FUNCTION_BLOCK PUBLIC RoutePlanner
VAR_INPUT
END_VAR
VAR_OUTPUT
END_VAR
VAR
	RejecLoadPosChoice			:       UINT :=5;
	RejectNextStationLocation	:		REAL;
	RejectNextStationIndex		:		BYTE;
	
	GoodULPosChoice				:       UINT :=5;
	GoodULNextStationLocation	:		REAL;
	GoodULNextStationIndex		:		BYTE;
	GoodFullCount : UINT := 0;
	PremiumFullCount : UINT := 0;
	GoodUL_1_NextStationFlag : BYTE := 5; // Next Station is defaulted to 5 ( reject)
	GoodUL_2_NextStationFlag : BYTE := 5; // Next Station is defaulted to 5 ( reject)
	GoodUL_3_NextStationFlag : BYTE := 5; // Next Station is defaulted to 5 ( reject)
	GoodUL_4_NextStationFlag : BYTE := 5; // Next Station is defaulted to 5 ( reject)
END_VAR

;

METHOD PUBLIC M_ExitCapInsertSta : BOOL
VAR_INPUT
	VehicleID		:	BYTE;
END_VAR
IF (PartsData.Status[VehicleID].OverallStatus <> ePartStatus.eReject AND 
    PartsData.Status[VehicleID].OverallStatus <> ePartStatus.eEmpty ) THEN  // we have a good part
   IF (LotsData.Lot.GoodUnloadEnabled) THEN // Good Unload is Enabled
		MoveToGoodUnload(VehicleID);
	ELSE // just go to reject
		MoveToReject(VehicleID);		
	END_IF		
ELSE  // we have a reject	
	MoveToReject(VehicleID);			
END_IF



(*

IF (PartsData.Status[VehicleID].OverallStatus = ePartStatus.eCapInserted) THEN
	Stations.fbVehicleManager[VehicleID].M_SetNextMoveParams(Pos:= MM_CONST.GOOD_UNLOAD_POS, Vel := 2.0, Acc := 2.0, StationIndex := MM_CONST.GOOD_UNLOAD_STA );
	Stations.fbVehicleManager[VehicleID].TriggerVehMov := TRUE;
ELSE 
	Stations.fbVehicleManager[VehicleID].M_SetNextMoveParams(Pos:= MM_CONST.REJECT_ULOAD_POS, Vel := 2.0, Acc := 2.0, StationIndex := MM_CONST.REJECT_ULOAD_STA );
 	Stations.fbVehicleManager[VehicleID].TriggerVehMov := TRUE;		
END_IF
*)

(*
Stations.fbVehicleManager[VehicleID].M_SetNextMoveParams(Pos:= MM_CONST.REJECT_ULOAD_POS, Vel := 2.0, Acc := 2.0, StationIndex := MM_CONST.REJECT_ULOAD_STA );
Stations.fbVehicleManager[VehicleID].TriggerVehMov := TRUE;
*)
END_METHOD

METHOD PUBLIC M_ExitGoodUnload : BOOL
VAR_INPUT
	VehicleID		:	BYTE;
END_VAR
MoveToReject(VehicleID);
END_METHOD

METHOD PUBLIC M_ExitGoodUnload_1 : BOOL
VAR_INPUT
	VehicleID		:	BYTE;
END_VAR
CASE GoodUL_1_NextStationFlag OF
	
    2:	
		MoveToGoodUnload_2(VehicleID);	
	
    3:
		MoveToGoodUnload_3(VehicleID);	
	
    4:
		MoveToGoodUnload_4(VehicleID);	
 
ELSE
		 MoveToReject(VehicleID);
	
END_CASE;
END_METHOD

METHOD PUBLIC M_ExitGoodUnload_2 : BOOL
VAR_INPUT
	VehicleID		:	BYTE;
END_VAR
CASE GoodUL_2_NextStationFlag OF
	
	
    3:
		MoveToGoodUnload_3(VehicleID);	
	
    4:
		MoveToGoodUnload_4(VehicleID);	
 
ELSE
		 MoveToReject(VehicleID);
	
END_CASE;
END_METHOD

METHOD PUBLIC M_ExitGoodUnload_3 : BOOL
VAR_INPUT
	VehicleID		:	BYTE;
END_VAR
CASE GoodUL_3_NextStationFlag OF
	

    4:
		MoveToGoodUnload_4(VehicleID);	
 
ELSE
		 MoveToReject(VehicleID);
	
END_CASE;
END_METHOD

METHOD PUBLIC M_ExitGoodUnload_4 : BOOL
VAR_INPUT
	VehicleID		:	BYTE;
END_VAR
MoveToReject(VehicleID);
END_METHOD

METHOD PUBLIC M_ExitIB_StopRobotClear : BOOL
VAR_INPUT
	VehicleID		:	BYTE;
END_VAR
IF (PartsData.Status[VehicleID].OverallStatus <> ePartStatus.eReject AND 
    PartsData.Status[VehicleID].OverallStatus <> ePartStatus.eEmpty ) THEN  // we have a good part
   IF (LotsData.Lot.CapInsertEnabled) THEN // Cap Is Enabled
		MoveToCap(VehicleID);
	ELSIF (LotsData.Lot.GoodUnloadEnabled) THEN // Good Unload is Enabled
		MoveToGoodUnload(VehicleID);
	ELSE // just go to reject
		MoveToReject(VehicleID);		
	END_IF		
ELSE  // we have a reject	
	MoveToReject(VehicleID);			
END_IF
END_METHOD

METHOD PUBLIC M_ExitLoad1Sta : BOOL
VAR_INPUT
	VehicleID		:	BYTE;
END_VAR
MoveToVision(VehicleID);
//MoveToStopBeforeVision(VehicleID);
END_METHOD

METHOD PUBLIC M_ExitLoad2Sta : BOOL
VAR_INPUT
	VehicleID		:	BYTE;
END_VAR
MoveToVision(VehicleID);
//MoveToStopBeforeVision(VehicleID);
END_METHOD

METHOD PUBLIC M_ExitLoad3Sta : BOOL
VAR_INPUT
	VehicleID		:	BYTE;
END_VAR
MoveToVision(VehicleID);
//MoveToStopBeforeVision(VehicleID);
END_METHOD

METHOD PUBLIC M_ExitLoad4Sta : BOOL
VAR_INPUT
	VehicleID		:	BYTE;
END_VAR
MoveToVision(VehicleID);
//MoveToStopBeforeVision(VehicleID);
END_METHOD

METHOD PUBLIC M_ExitPistonInsertSta : BOOL
VAR_INPUT
	VehicleID		:	BYTE;
END_VAR
IF (PartsData.Status[VehicleID].OverallStatus <> ePartStatus.eReject AND 
    PartsData.Status[VehicleID].OverallStatus <> ePartStatus.eEmpty ) THEN  // we have a good part
    IF (Stations.fbLoad1Sta.HoldVehicle_IBStop) THEN //Yushin wants to load 
		MoveToIBStopRobotClear(VehicleID);
	ELSIF (LotsData.Lot.CapInsertEnabled) THEN // Cap Is Enabled
		MoveToCap(VehicleID);
	ELSIF (LotsData.Lot.GoodUnloadEnabled) THEN // Good Unload is Enabled
		MoveToGoodUnload(VehicleID);
	ELSE // just go to reject
		MoveToReject(VehicleID);		
	END_IF		
ELSE  // we have a reject	
	IF (Stations.fbLoad1Sta.HoldVehicle_IBStop) THEN //Yushin wants to load 
		MoveToIBStopRobotClear(VehicleID);
	ELSE  // just go to reject
		MoveToReject(VehicleID);			
	END_IF
END_IF

(*
IF (Stations.fbLoad1Sta.HoldVehicle_IBStop) THEN //Yushin wants to load 
	Stations.fbVehicleManager[VehicleID].M_SetNextMoveParams(Pos:= MM_CONST.IB_STOP_ROBOT_CLEAR_POS, Vel := 2.0, Acc := 2.0, StationIndex := MM_CONST.IB_STOP_ROBOT_CLEAR_STA );
	Stations.fbVehicleManager[VehicleID].TriggerVehMov := TRUE;
ELSE // move straight to the cap station or reject based on part status
    IF (PartsData.Status[VehicleID].OverallStatus = ePartStatus.ePistonInserted) THEN
		 Stations.fbVehicleManager[VehicleID].M_SetNextMoveParams(Pos:= MM_CONST.CAP_POS, Vel := 2.0, Acc := 2.0, StationIndex := MM_CONST.CAP_STA );
		 Stations.fbVehicleManager[VehicleID].TriggerVehMov := TRUE;
	ELSE 
		Stations.fbVehicleManager[VehicleID].M_SetNextMoveParams(Pos:= MM_CONST.REJECT_ULOAD_POS, Vel := 2.0, Acc := 2.0, StationIndex := MM_CONST.REJECT_ULOAD_STA );
 		Stations.fbVehicleManager[VehicleID].TriggerVehMov := TRUE;
	END_IF
   
END_IF



//Stations.fbVehicleManager[VehicleID].M_SetNextMoveParams(Pos:= MM_CONST.CAP_POS, Vel := 2.0, Acc := 2.0, StationIndex := MM_CONST.CAP_STA );
//Stations.fbVehicleManager[VehicleID].TriggerVehMov := TRUE;


// Stations.fbVehicleManager[VehicleID].M_SetNextMoveParams(Pos:= MM_CONST.REJECT_ULOAD_POS, Vel := 2.0, Acc := 2.0, StationIndex := MM_CONST.REJECT_ULOAD_STA );
 // Stations.fbVehicleManager[VehicleID].TriggerVehMov := TRUE;


(*

	Stations.fbVehicleManager[VehicleID].M_SetNextMoveParams(Pos:= MM_CONST.PISTON_POS, Vel := 2.0, Acc := 2.0, StationIndex := MM_CONST.PISTON_STA );
	Stations.fbVehicleManager[VehicleID].TriggerVehMov := TRUE;
	*)

(*


IF (Stations.fbLoad1Sta.HoldVehicle_IBStop) THEN //Yushin wants to load 
	Stations.fbVehicleManager[VehicleID].M_SetNextMoveParams(Pos:= MM_CONST.IB_STOP_ROBOT_CLEAR_POS, Vel := 2.0, Acc := 2.0, StationIndex := MM_CONST.IB_STOP_ROBOT_CLEAR_STA );
	Stations.fbVehicleManager[VehicleID].TriggerVehMov := TRUE;
ELSE // move straight to the cap station
	// NEED TO REMOVE THIS AFTER DEBUG ON 3/19/2017... WE ARE BYPASSING CAP STATION FOR NOW 
    //Stations.fbVehicleManager[VehicleID].M_SetNextMoveParams(Pos:= MM_CONST.CAP_POS, Vel := 2.0, Acc := 2.0, StationIndex := MM_CONST.CAP_STA );
	//Stations.fbVehicleManager[VehicleID].TriggerVehMov := TRUE;
	
	Stations.fbVehicleManager[VehicleID].M_SetNextMoveParams(Pos:= MM_CONST.GOOD_UNLOAD_POS, Vel := 2.0, Acc := 2.0, StationIndex := MM_CONST.GOOD_UNLOAD_STA );
	Stations.fbVehicleManager[VehicleID].TriggerVehMov := TRUE;
			
END_IF

*)
*)
END_METHOD

METHOD PUBLIC M_ExitRejectUnload : BOOL
VAR_INPUT	
	VehicleID		:	BYTE;
END_VAR
RejecLoadPosChoice := RejecLoadPosChoice -1; //we initialize with this variable as 5;
IF (RejecLoadPosChoice<=0 OR RejecLoadPosChoice>=4 ) THEN 
	RejecLoadPosChoice := 4;
END_IF
CASE RejecLoadPosChoice OF
				4: 
					RejectNextStationLocation := MM_CONST.OB_STOP_ROBOT_CLEAR_POS;
					RejectNextStationIndex	:= MM_CONST.OB_STOP_ROBOT_CLEAR_STA;
				3:
					RejectNextStationLocation := MM_CONST.LOAD_3_POS;
					RejectNextStationIndex	:= MM_CONST.LOAD_3_STA;
				2:
					RejectNextStationLocation := MM_CONST.LOAD_2_POS;
					RejectNextStationIndex	:= MM_CONST.LOAD_2_STA;
				1:
					RejectNextStationLocation := MM_CONST.LOAD_1_POS;
					RejectNextStationIndex	:= MM_CONST.LOAD_1_STA;						
END_CASE				
	
Stations.fbVehicleManager[VehicleID].M_SetNextMoveParams(Pos:= RejectNextStationLocation, Vel := 2.0, Acc := 2.0, StationIndex := RejectNextStationIndex );
Stations.fbVehicleManager[VehicleID].TriggerVehMov := TRUE;
END_METHOD

METHOD PUBLIC M_ExitVisionSta : BOOL
VAR_INPUT
	VehicleID		:	BYTE;
END_VAR
IF (PartsData.Status[VehicleID].OverallStatus <> ePartStatus.eReject AND 
    PartsData.Status[VehicleID].OverallStatus <> ePartStatus.eEmpty ) THEN  // we have a good part
    IF (LotsData.Lot.PistonInsertEnabled) THEN //Piston is enabled
		MoveToPiston(VehicleID);
	ELSIF (Stations.fbLoad1Sta.HoldVehicle_IBStop) THEN //Yushin wants to load 
		MoveToIBStopRobotClear(VehicleID);
	ELSIF (LotsData.Lot.CapInsertEnabled) THEN // If Cap Is Enabled
		MoveToCap(VehicleID);		
	ELSIF (LotsData.Lot.GoodUnloadEnabled) THEN // If Good Unload is Enabled
		MoveToGoodUnload(VehicleID);
	ELSE // just go to reject
		MoveToReject(VehicleID);	
	END_IF		
ELSE  // we have a reject	
	IF (Stations.fbLoad1Sta.HoldVehicle_IBStop) THEN //Yushin wants to load 
		MoveToIBStopRobotClear(VehicleID);
	ELSE  // just go to reject
		MoveToReject(VehicleID);		
	END_IF
END_IF
END_METHOD

METHOD PUBLIC M_NotifyVehStaCmpl : BOOL
VAR_INPUT
	StationIndex 	:	BYTE;
	VehicleID		:	BYTE;
END_VAR
CASE StationIndex OF

		
	MM_CONST.LOAD_1_STA:
        M_ExitLoad1Sta(VehicleID := VehicleID);

    MM_CONST.LOAD_2_STA:
		M_ExitLoad2Sta(VehicleID := VehicleID);

    MM_CONST.LOAD_3_STA:
		M_ExitLoad3Sta(VehicleID := VehicleID);			

    MM_CONST.LOAD_4_STA:					
       M_ExitLoad4Sta(VehicleID := VehicleID);

    MM_CONST.STOP_BEFORE_VISION_STA:
		M_OBExit_StopBeforeVision(VehicleID := VehicleID);

    MM_CONST.VISION_STA:
		M_ExitVisionSta(VehicleID := VehicleID);

    MM_CONST.PISTON_STA:		
		M_ExitPistonInsertSta(VehicleID := VehicleID);

	MM_CONST.IB_STOP_ROBOT_CLEAR_STA:
		M_ExitIB_StopRobotClear(VehicleID := VehicleID);
    
    MM_CONST.CAP_STA:
		M_ExitCapInsertSta(VehicleID := VehicleID);
   
    MM_CONST.GOOD_UNLOAD_STA:	
	   M_ExitGoodUnload(VehicleID:=VehicleID);  

    MM_CONST.GOOD_UL_1_STA:
		M_ExitGoodUnload_1(VehicleID:=VehicleID); 
	
	MM_CONST.GOOD_UL_2_STA:
		M_ExitGoodUnload_2(VehicleID:=VehicleID); 
		
	MM_CONST.GOOD_UL_3_STA:
		M_ExitGoodUnload_3(VehicleID:=VehicleID); 
	
	MM_CONST.GOOD_UL_4_STA:	
		M_ExitGoodUnload_4(VehicleID:=VehicleID); 
  

    MM_CONST.REJECT_ULOAD_STA:		
		M_ExitRejectUnload(VehicleID:= VehicleID);
	
	MM_CONST.OB_STOP_ROBOT_CLEAR_STA:
		M_OBExitOB_StopBeforeRobotClear(VehicleID := VehicleID);

ELSE; 
END_CASE
END_METHOD

METHOD PUBLIC M_OBExit_StopBeforeVision : BOOL
VAR_INPUT
	VehicleID		:	BYTE;
END_VAR
IF (PartsData.Status[VehicleID].OverallStatus = ePartStatus.eEmpty) THEN
  MoveToReject(VehicleID);
ELSE	
    MoveToVision(VehicleID);
END_IF
END_METHOD

METHOD PUBLIC M_OBExitOB_StopBeforeRobotClear : BOOL
VAR_INPUT
	VehicleID: BYTE;
END_VAR
MoveToLoadPos4(VehicleID);
END_METHOD

METHOD PUBLIC MoveToCap : BOOL
VAR_INPUT
	VehicleID		:	BYTE;
END_VAR
Stations.fbVehicleManager[VehicleID].M_SetNextMoveParams(Pos:= MM_CONST.CAP_POS, Vel := 2.0, Acc := 2.0, StationIndex := MM_CONST.CAP_STA );
Stations.fbVehicleManager[VehicleID].TriggerVehMov := TRUE;
END_METHOD

METHOD PUBLIC MoveToGoodUnload : BOOL
VAR_INPUT
	VehicleID		:	BYTE;
END_VAR
// If for some reason a reject parts comes here, send it to reject station
	IF (PartsData.Status[VehicleID].OverallStatus = ePartStatus.eReject) THEN
		MoveToReject(VehicleID);
		RETURN; 
	END_IF	

// If the Auto-Bagger is not enabled, then we distribute the pallets to all 2 UL stations 

IF (NOT LotsData.Lot.AutoBaggerEnabled) THEN
	IF (PartsData.Status[VehicleID].Premium) THEN
		MoveToGoodUnload_2(VehicleID);
	ELSIF (PartsData.Status[VehicleID].Good) THEN
        MoveToGoodUnload_3(VehicleID);
	ELSE
		MoveToReject(VehicleID);
	END_IF
	
		// Reset all Chute Part Counters 
	Config.PremiumCount1 := 0;
	Config.PremiumCount2 := 0;
	Config.GoodCount1 := 0;
	Config.GoodCount2 := 0;
	GoodFullCount := 0;
    PremiumFullCount := 0;
	
	// Exit from this routine
	RETURN;
END_IF
 
// If Auto-bagger is enabled  
// Chute choice is relegated at the individual station
IF (PartsData.Status[VehicleID].Premium) THEN
	MoveToGoodUnload_1(VehicleID);	
ELSIF (PartsData.Status[VehicleID].Good) THEN
	MoveToGoodUnload_3(VehicleID);
ELSE
	MoveToReject(VehicleID);
END_IF

(*
IF (PartsData.Status[VehicleID].Premium) THEN
	    // First preference is to fill Chute closest to Reject Station. 
		IF((Config.PremiumCount1 < LotsData.Lot.QuantityInBag) AND ((Config.PremiumCount2 < (LotsData.Lot.QuantityInBag-10)) OR (Config.PremiumCount2 = LotsData.Lot.QuantityInBag))) THEN
			MoveToGoodUnload_1(VehicleID);			
			PremiumFullCount := 0;
		ELSIF (Config.PremiumCount2 < LotsData.Lot.QuantityInBag) THEN
			MoveToGoodUnload_2(VehicleID);			
			PremiumFullCount := 0;
		ELSE  // demote the status of the parts to Good
			PartsData.Status[VehicleID].Premium := FALSE;
			PartsData.Status[VehicleID].Good := TRUE;
			PremiumFullCount := PremiumFullCount + 1;
		END_IF
	END_IF

// If the Parts are Good 	
	IF (PartsData.Status[VehicleID].Good) THEN   
		//First preference is to fill the Chute downstream closer to reject/premium 
		IF ((Config.GoodCount1 < LotsData.Lot.QuantityInBag) AND ((Config.GoodCount2 < (LotsData.Lot.QuantityInBag-10)) OR (Config.GoodCount2 = LotsData.Lot.QuantityInBag))) THEN
			MoveToGoodUnload_3(VehicleID);	
			GoodFullCount := 0;
		ELSIF (Config.GoodCount2 < LotsData.Lot.QuantityInBag) THEN
			MoveToGoodUnload_4(VehicleID);	
			GoodFullCount := 0;
		ELSE
			PartsData.Status[VehicleID].Premium := FALSE;
			PartsData.Status[VehicleID].Good := FALSE;
			PartsData.Status[VehicleID].OverallStatus := ePartStatus.eReject;
			PartsData.Status[VehicleID].GoodUnload := FALSE;
			GoodFullCount := GoodFullCount + 1;
		END_IF	
	END_IF
    	
	IF (PartsData.Status[VehicleID].OverallStatus = ePartStatus.eReject) THEN
		MoveToReject(VehicleID);
	END_IF	
	
	IF (GoodFullCount >= 5 OR PremiumFullCount >= 5) THEN
		Stations.fbCycleControl.StopRequested := TRUE;
		Status.AutoBaggerStatusMsg := 'AutoBagger: No drop location available. Clear Chutes';
	END_IF	
	
*)
END_METHOD

METHOD PUBLIC MoveToGoodUnload_1 : BOOL
VAR_INPUT
	VehicleID		:	BYTE;
END_VAR
Stations.fbVehicleManager[VehicleID].M_SetNextMoveParams(Pos:= MM_CONST.GOOD_UL_1_POS, Vel := 2.0, Acc := 2.0, StationIndex := MM_CONST.GOOD_UL_1_STA );
Stations.fbVehicleManager[VehicleID].TriggerVehMov := TRUE;
END_METHOD

METHOD PUBLIC MoveToGoodUnload_2 : BOOL
VAR_INPUT
	VehicleID		:	BYTE;
END_VAR
Stations.fbVehicleManager[VehicleID].M_SetNextMoveParams(Pos:= MM_CONST.GOOD_UL_2_POS, Vel := 2.0, Acc := 2.0, StationIndex := MM_CONST.GOOD_UL_2_STA );
Stations.fbVehicleManager[VehicleID].TriggerVehMov := TRUE;
END_METHOD

METHOD PUBLIC MoveToGoodUnload_3 : BOOL
VAR_INPUT
	VehicleID		:	BYTE;
END_VAR
Stations.fbVehicleManager[VehicleID].M_SetNextMoveParams(Pos:= MM_CONST.GOOD_UL_3_POS, Vel := 2.0, Acc := 2.0, StationIndex := MM_CONST.GOOD_UL_3_STA );
Stations.fbVehicleManager[VehicleID].TriggerVehMov := TRUE;
END_METHOD

METHOD PUBLIC MoveToGoodUnload_4 : BOOL
VAR_INPUT
	VehicleID		:	BYTE;
END_VAR
Stations.fbVehicleManager[VehicleID].M_SetNextMoveParams(Pos:= MM_CONST.GOOD_UL_4_POS, Vel := 2.0, Acc := 2.0, StationIndex := MM_CONST.GOOD_UL_4_STA );
Stations.fbVehicleManager[VehicleID].TriggerVehMov := TRUE;
END_METHOD

METHOD PUBLIC MoveToIBStopRobotClear : BOOL
VAR_INPUT
	VehicleID		:	BYTE;
END_VAR
Stations.fbVehicleManager[VehicleID].M_SetNextMoveParams(Pos:= MM_CONST.IB_STOP_ROBOT_CLEAR_POS, Vel := 2.0, Acc := 2.0, StationIndex := MM_CONST.IB_STOP_ROBOT_CLEAR_STA );
Stations.fbVehicleManager[VehicleID].TriggerVehMov := TRUE;
END_METHOD

METHOD PUBLIC MoveToLoadPos4 : BOOL
VAR_INPUT
	VehicleID		:	BYTE;
END_VAR
Stations.fbVehicleManager[VehicleID].M_SetNextMoveParams(Pos:= MM_CONST.LOAD_4_POS, Vel := 2.0, Acc := 2.0, StationIndex := MM_CONST.LOAD_4_STA );
Stations.fbVehicleManager[VehicleID].TriggerVehMov := TRUE;
END_METHOD

METHOD PUBLIC MoveToPiston : BOOL
VAR_INPUT
	VehicleID		:	BYTE;
END_VAR
Stations.fbVehicleManager[VehicleID].M_SetNextMoveParams(Pos:= MM_CONST.PISTON_POS, Vel := 2.0, Acc := 2.0, StationIndex := MM_CONST.PISTON_STA );
Stations.fbVehicleManager[VehicleID].TriggerVehMov := TRUE;
END_METHOD

METHOD PUBLIC MoveToReject : BOOL
VAR_INPUT
	VehicleID		:	BYTE;
END_VAR
Stations.fbVehicleManager[VehicleID].M_SetNextMoveParams(Pos:= MM_CONST.REJECT_ULOAD_POS, Vel := 2.0, Acc := 2.0, StationIndex := MM_CONST.REJECT_ULOAD_STA );
Stations.fbVehicleManager[VehicleID].TriggerVehMov := TRUE;
END_METHOD

METHOD PUBLIC MoveToStopBeforeVision : BOOL
VAR_INPUT
	VehicleID		:	BYTE;
END_VAR
Stations.fbVehicleManager[VehicleID].M_SetNextMoveParams(Pos:= MM_CONST.STOP_BEFORE_VISION_POS, Vel := 2.0, Acc := 0.5, StationIndex := MM_CONST.STOP_BEFORE_VISION_STA);
Stations.fbVehicleManager[VehicleID].TriggerVehMov := TRUE;
END_METHOD

METHOD PUBLIC MoveToVision : BOOL
VAR_INPUT
	VehicleID		:	BYTE;
END_VAR
Stations.fbVehicleManager[VehicleID].M_SetNextMoveParams(Pos:= MM_CONST.VISION_POS, Vel := 2.0, Acc := 2.0, StationIndex := MM_CONST.VISION_STA );
Stations.fbVehicleManager[VehicleID].TriggerVehMov := TRUE;
END_METHOD

PROPERTY PUBLIC P_GoodUnload_1_NextStaFlag : BYTE
SET
GoodUL_1_NextStationFlag := P_GoodUnload_1_NextStaFlag;
END_SET
END_PROPERTY

PROPERTY PUBLIC P_GoodUnload_2_NextStaFlag : BYTE
SET
GoodUL_2_NextStationFlag := P_GoodUnload_2_NextStaFlag;
END_SET
END_PROPERTY

PROPERTY PUBLIC P_GoodUnload_3_NextStaFlag : BYTE
SET
GoodUL_3_NextStationFlag := P_GoodUnload_3_NextStaFlag;
END_SET
END_PROPERTY

PROPERTY PUBLIC P_GoodUnload_4_NextStaFlag : BYTE
SET
GoodUL_4_NextStationFlag := P_GoodUnload_4_NextStaFlag;
END_SET
END_PROPERTY

METHOD SetGoodULLoadPosChoiceToInit : BOOL
VAR_INPUT
END_VAR
GoodULPosChoice	:=5;
END_METHOD

METHOD PUBLIC SetRejectLoadPosChoiceToInit : BOOL
VAR_INPUT
END_VAR
RejecLoadPosChoice := 5;
END_METHOD

END_FUNCTION_BLOCK

(* stored: Version 1.1.0.1, ProductVersion 3.1.4022.6
   POU RoutePlanner: Id {1695e7c5-e1de-4f29-9ed6-9e8b7377b48c}, SpecialFunc None
   Folder CmdsForMM: Id {5d9d421f-970e-42e1-8a42-92df3faf0379}
   Method M_ExitCapInsertSta: Id {8d622e34-31a9-4b99-833a-aad5e6f895d3}
   Method M_ExitGoodUnload: Id {c40521b2-5dfd-42b8-8190-74370c4d9b2a}
   Method M_ExitGoodUnload_1: Id {88fd2d1b-ecf2-4ff9-a23e-78d77c0aee7e}
   Method M_ExitGoodUnload_2: Id {a9d07807-873b-4013-9d12-eba4686a962d}
   Method M_ExitGoodUnload_3: Id {1851bf7e-7d63-43ee-8dd0-fa5d46c5268b}
   Method M_ExitGoodUnload_4: Id {259f11c1-8cdb-4aa8-b0b8-f78198557539}
   Method M_ExitIB_StopRobotClear: Id {200d0821-42b0-4224-8914-cb06fec18d9b}
   Method M_ExitLoad1Sta: Id {1e96eb00-4803-45e3-a722-ffc4394e0e30}
   Method M_ExitLoad2Sta: Id {80ecc0a6-16af-42d6-afca-f6706e1a2a1a}
   Method M_ExitLoad3Sta: Id {33284259-7360-4d69-8a2c-c0431b108cfd}
   Method M_ExitLoad4Sta: Id {32758d78-a5e0-42e4-931d-cd1fe71e0025}
   Method M_ExitPistonInsertSta: Id {56dc8c6b-ccb3-4434-9451-a97b46c9faeb}
   Method M_ExitRejectUnload: Id {ccb65de4-bcfb-4fc1-8aac-37c1010e4f7e}
   Method M_ExitVisionSta: Id {460c3f27-2d5d-4cf0-980d-e3f28721f258}
   Method M_NotifyVehStaCmpl: Id {dcb99565-f67f-4080-8f23-9f88067292d8}
   Method M_OBExit_StopBeforeVision: Id {f4664737-0532-442c-84e9-a8acd492192b}
   Method M_OBExitOB_StopBeforeRobotClear: Id {ef907099-4308-412f-b9da-3a5773808998}
   Method MoveToCap: Id {b3a3c957-df72-41f2-aa94-e9454f901db0}
   Method MoveToGoodUnload: Id {dd6d7f40-5483-4dab-a0b1-2dfc52726873}
   Method MoveToGoodUnload_1: Id {036b2203-da67-4b56-b00c-820db31800c4}
   Method MoveToGoodUnload_2: Id {217b4eef-b729-4c7f-b6ef-b1d6e9f68814}
   Method MoveToGoodUnload_3: Id {7dbe0160-e4b3-41b5-a112-53aa9fa94373}
   Method MoveToGoodUnload_4: Id {0b3ad729-bf0d-4b82-b48e-ecfa284451f6}
   Method MoveToIBStopRobotClear: Id {bfdaf3c0-099b-4e3a-a3a0-d4cba0ed7cb1}
   Method MoveToLoadPos4: Id {8d73af71-127f-4216-a753-2bc8f5e84513}
   Method MoveToPiston: Id {b6478e91-3e94-418e-8223-766a60db7c7a}
   Method MoveToReject: Id {3158e929-675b-4d83-8335-ae0442af3432}
   Method MoveToStopBeforeVision: Id {386d9d5a-0a88-4168-aff5-6a35e5cbc83b}
   Method MoveToVision: Id {1a0dd900-73ca-449f-8f17-2f4fca9622f9}
   Property P_GoodUnload_1_NextStaFlag: Id {f9e7abad-60f2-4976-9845-8db03eea03d8}
   Set Set: Id {c9cc38cf-e9e4-4452-8589-d5038e08fdb8}
   Property P_GoodUnload_2_NextStaFlag: Id {7f80488f-9639-4f42-8544-e6f7b23f08fb}
   Set Set: Id {56a96b89-21db-40c3-b276-04beab588c30}
   Property P_GoodUnload_3_NextStaFlag: Id {d12314e0-0fd8-4c5e-ac6c-bc307a863cef}
   Set Set: Id {1bae7f06-aaef-415e-a758-f37fd0d693c0}
   Property P_GoodUnload_4_NextStaFlag: Id {494ff4bb-7954-415b-b866-1846e8175cfd}
   Set Set: Id {b7dd0c84-7634-4163-ad9e-a1ce11141e97}
   Method SetGoodULLoadPosChoiceToInit: Id {8f29e26a-fcd3-4639-b579-551bfb92c1d2}
   Method SetRejectLoadPosChoiceToInit: Id {ea023fca-5e90-4160-ae8d-2874f107f690} *)
